{region '#Template'}
	{attribute 'Version' := '5.1.0.0'}
	{attribute 'Tags' := '"LCID": "1031", "Text": "RA, HC, Controller"'}
	{attribute 'Tags' := '"LCID": "1033", "Text": "RA, HC, Controller"'}
	{attribute 'Using' := '"Type": "Template", "URI": "BA2_Param"'}
	{attribute 'Description' := '"LCID": "1031", "Text": "Heiz-/Kühlregelung Raum"'}
	{attribute 'Description' := '"LCID": "1033", "Text": "Heating-/cooling-controller room"'}
{endregion}
FUNCTION_BLOCK FB_BA_HeatCool_PID EXTENDS FB_BA_Ext_HeatCoolBase         		
VAR_INPUT    		
	bPrc							: BOOL;				// presence-detector
	bWdwCon							: BOOL;				// window-contact - TRUE = OPEN
	eMedium							: E_BA_Medium;		// actual medium when using 2-pipe-system: heating or cooling
	bDewPnt							: BOOL;				// dew-point-detector - TRUE = ALARM
	fRmT							: REAL;				// actual room-temperature
	fRmTAdj							: REAL;				// manual adjustment of room-temperature, if desired.
	stBuildingSpRmT					: ST_BA_SpRmT;		// set points for all energy levels
	eBuildingEnergyLevel			: E_BA_EnergyLvlEx;	// current energy levels
	                                                    
END_VAR             			                        
VAR_OUTPUT          	                                
	bCtrlHtgActv					: BOOL;				// controller heating is active	
	fCtrlValHtg						: REAL;				// control-value heating
	bCtrlColActv					: BOOL;				// controller cooling is active	
	fCtrlValCol						: REAL;				// control-value cooling
	eReqdMedium						: E_BA_Medium;		// requested medium
END_VAR                                                 
VAR_INPUT CONSTANT PERSISTENT                           
	ePipeSys						: E_BA_PipeSys;		// selection 2-pipe or 4-pipe system
	{attribute 'parameterUnit':= 's'}                   
	nFnctSelChgOvrDly 				: UDINT;			// switch-over-delay from heating to cooling or vice versa	
	fRmTAdjLimit					: REAL;				// positive and negative limit of room temperature adjust value
END_VAR                  		
VAR_INPUT CONSTANT
	CtrlHtg							: FB_BA_Loop;
	CtrlCol							: FB_BA_Loop;
END_VAR
VAR
	RmTAdj							: FB_BA_RmTAdj;
	EnergLvlSlcn					: FB_BA_PrioSwi_UDI04;
	SpSlcnHtg						: FB_BA_MUX_R04;
	SpSclnCol						: FB_BA_MUX_R04;
	FnctSel							: FB_BA_FnctSel;
	RmTAdjSel						: FB_BA_LastWriterWins_R04;
	fRmTAdjLimited					: REAL;		// limited room temperature adjust value
END_VAR
VAR // added by the converter: edge detectors and wires of the graphical bodies
    _w1 : REAL;
END_VAR

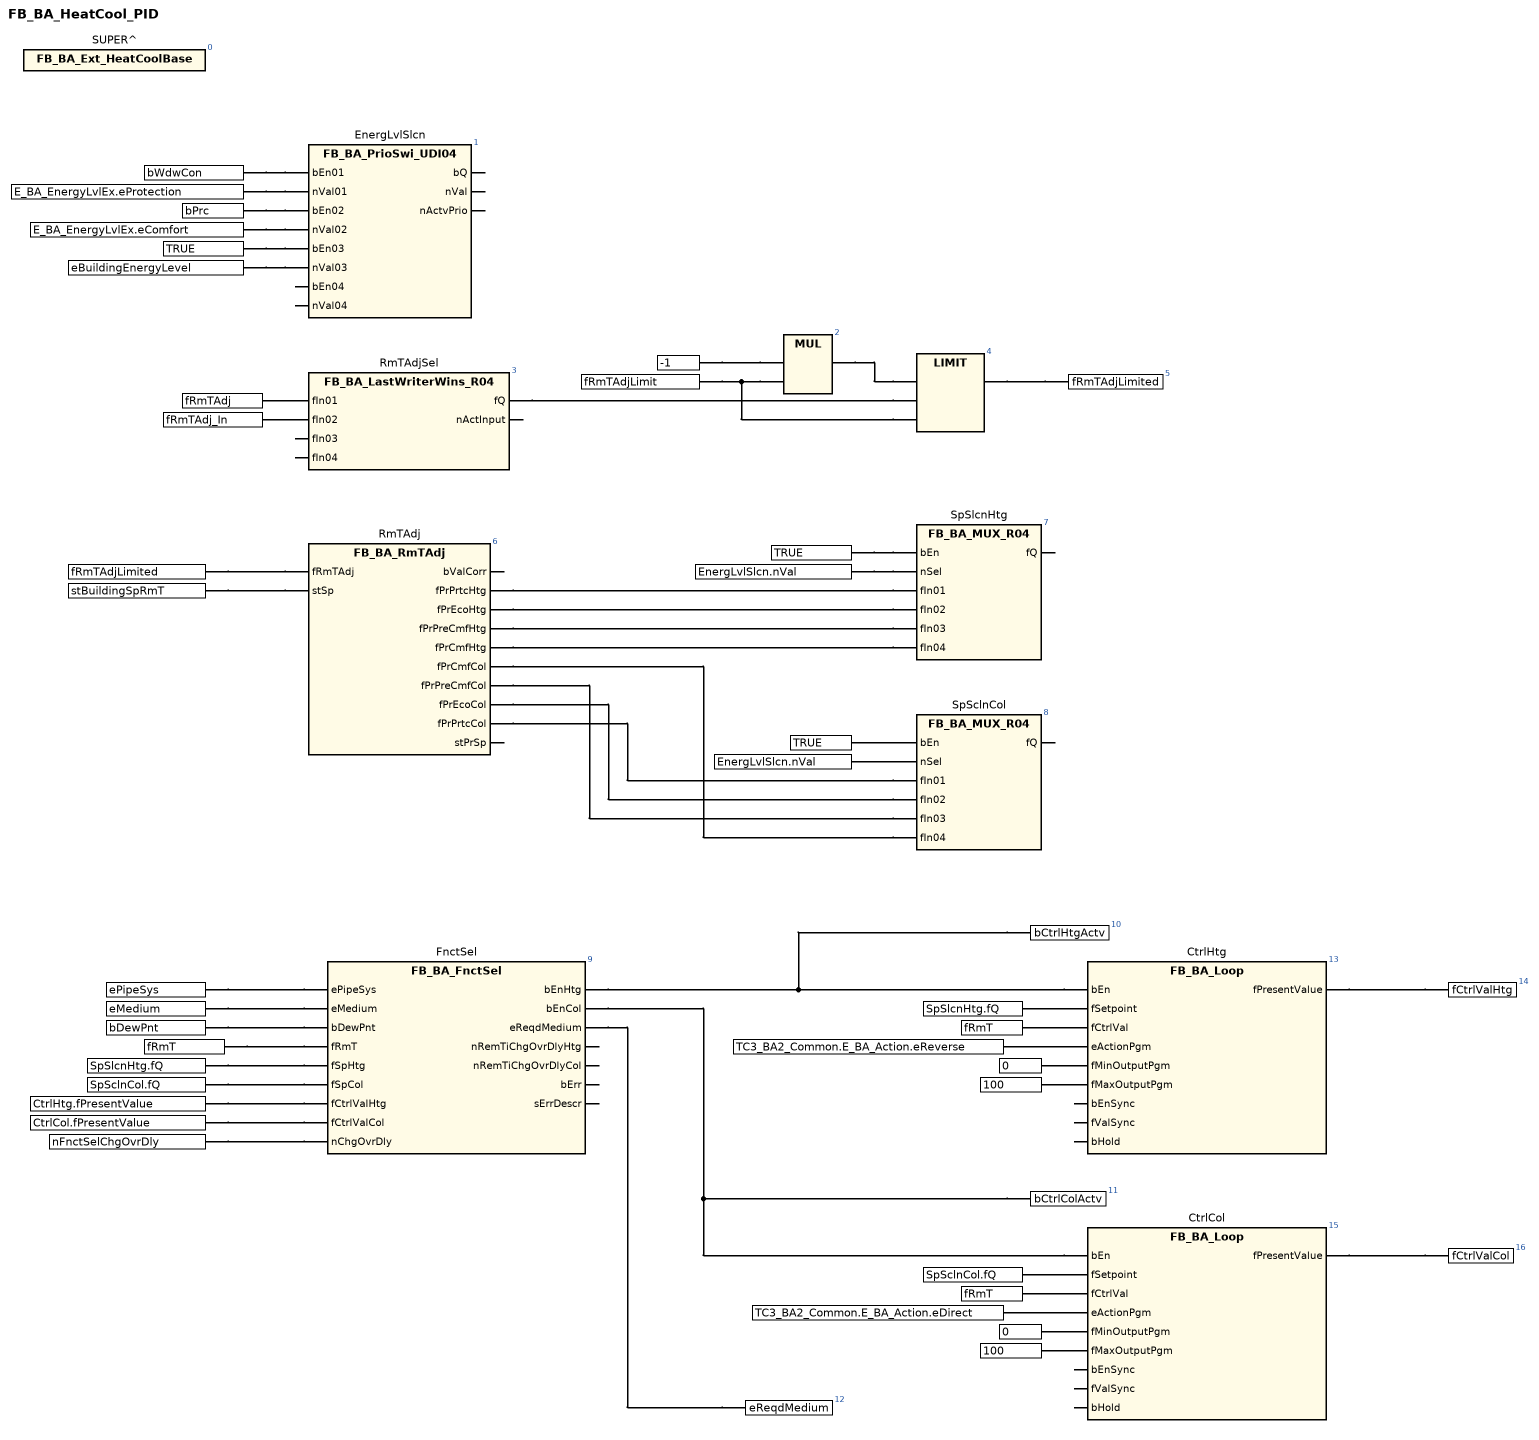
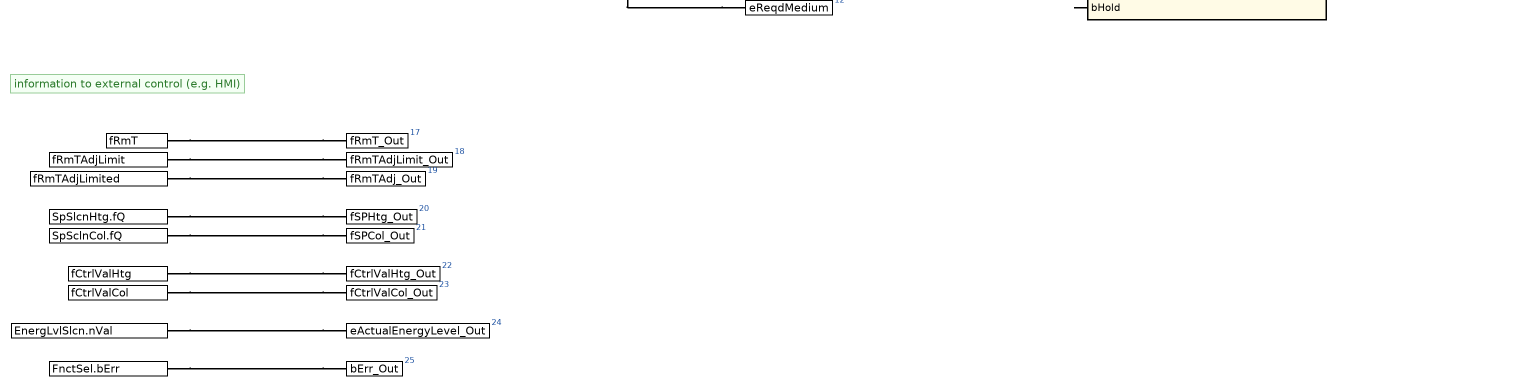
SUPER^(); // FB_BA_Ext_HeatCoolBase
EnergLvlSlcn(
    bEn01 := bWdwCon,
    nVal01 := E_BA_EnergyLvlEx.eProtection,
    bEn02 := bPrc,
    nVal02 := E_BA_EnergyLvlEx.eComfort,
    bEn03 := TRUE,
    nVal03 := eBuildingEnergyLevel); // FB_BA_PrioSwi_UDI04
_w1 := -1 * fRmTAdjLimit;
RmTAdjSel(fIn01 := fRmTAdj, fIn02 := fRmTAdj_In); // FB_BA_LastWriterWins_R04
fRmTAdjLimited := LIMIT(_w1, RmTAdjSel.fQ, fRmTAdjLimit);
RmTAdj(fRmTAdj := fRmTAdjLimited, stSp := stBuildingSpRmT); // FB_BA_RmTAdj
SpSlcnHtg(
    bEn := TRUE,
    nSel := EnergLvlSlcn.nVal,
    fIn01 := RmTAdj.fPrPrtcHtg,
    fIn02 := RmTAdj.fPrEcoHtg,
    fIn03 := RmTAdj.fPrPreCmfHtg,
    fIn04 := RmTAdj.fPrCmfHtg); // FB_BA_MUX_R04
SpSclnCol(
    bEn := TRUE,
    nSel := EnergLvlSlcn.nVal,
    fIn01 := RmTAdj.fPrPrtcCol,
    fIn02 := RmTAdj.fPrEcoCol,
    fIn03 := RmTAdj.fPrPreCmfCol,
    fIn04 := RmTAdj.fPrCmfCol); // FB_BA_MUX_R04
FnctSel(
    ePipeSys := ePipeSys,
    eMedium := eMedium,
    bDewPnt := bDewPnt,
    fRmT := fRmT,
    fSpHtg := SpSlcnHtg.fQ,
    fSpCol := SpSclnCol.fQ,
    fCtrlValHtg := CtrlHtg.fPresentValue,
    fCtrlValCol := CtrlCol.fPresentValue,
    nChgOvrDly := nFnctSelChgOvrDly); // FB_BA_FnctSel
bCtrlHtgActv := FnctSel.bEnHtg;
bCtrlColActv := FnctSel.bEnCol;
eReqdMedium := FnctSel.eReqdMedium;
CtrlHtg(
    bEn := FnctSel.bEnHtg,
    fSetpoint := SpSlcnHtg.fQ,
    fCtrlVal := fRmT,
    eActionPgm := TC3_BA2_Common.E_BA_Action.eReverse,
    fMinOutputPgm := 0,
    fMaxOutputPgm := 100); // FB_BA_Loop
fCtrlValHtg := CtrlHtg.fPresentValue;
CtrlCol(
    bEn := FnctSel.bEnCol,
    fSetpoint := SpSclnCol.fQ,
    fCtrlVal := fRmT,
    eActionPgm := TC3_BA2_Common.E_BA_Action.eDirect,
    fMinOutputPgm := 0,
    fMaxOutputPgm := 100); // FB_BA_Loop
fCtrlValCol := CtrlCol.fPresentValue;
// information to external control (e.g. HMI)
fRmT_Out := fRmT;
fRmTAdjLimit_Out := fRmTAdjLimit;
fRmTAdj_Out := fRmTAdjLimited;
fSPHtg_Out := SpSlcnHtg.fQ;
fSPCol_Out := SpSclnCol.fQ;
fCtrlValHtg_Out := fCtrlValHtg;
fCtrlValCol_Out := fCtrlValCol;
eActualEnergyLevel_Out := EnergLvlSlcn.nVal;
bErr_Out := FnctSel.bErr;

METHOD FB_init : BOOL
VAR_INPUT
	bInitRetains : BOOL; // if TRUE, the retain variables are initialized (warm start / cold start)
	bInCopyCode : BOOL;  // if TRUE, the instance afterwards gets moved into the copy code (online change)
END_VAR
ePipeSys							:= E_BA_PipeSys.e4Pipe;	// selection 2-pipe or 4-pipe system
nFnctSelChgOvrDly 					:= 120;					// switch-over-delay [s] from heating to cooling or vice versa	
fRmTAdjLimit						:= 1;					// positive and negative limit of room temperature adjust value

CtrlHtg.iParent						:= THIS^;
CtrlHtg.iLabel						:= LblCtl_RoomTemperatureControl;
CtrlHtg.eOpMode						:= E_BA_PIDMode.ePID;								 	 										 
CtrlHtg.eOutputUnit					:= E_BA_Unit.eOther_Percent;
CtrlHtg.fProportionalConstant		:= 3;
CtrlHtg.fIntegralConstant			:= 180;
CtrlHtg.fDerivativeConstant			:= 0;
CtrlHtg.fCOVIncrement				:= 0;
CtrlHtg.nDampConstant				:= 0;
CtrlHtg.fNeutralZone				:= 0;

CtrlCol.iParent						:= THIS^;
CtrlCol.iLabel						:= LblCtl_RoomTemperatureControl;
CtrlCol.eOpMode						:= E_BA_PIDMode.ePID;								 	 										 
CtrlCol.eOutputUnit					:= E_BA_Unit.eOther_Percent;
CtrlCol.fProportionalConstant		:= 3;
CtrlCol.fIntegralConstant			:= 180;
CtrlCol.fDerivativeConstant			:= 0;
CtrlCol.fCOVIncrement				:= 0;
CtrlCol.nDampConstant				:= 0;
CtrlCol.fNeutralZone				:= 0;
END_METHOD

END_FUNCTION_BLOCK

(* stored: Version 1.1.0.1, ProductVersion 3.1.4024.15
   POU FB_BA_HeatCool_PID: Id {c0e37cb5-7965-4a23-a2cd-66b383c1dd05}, SpecialFunc None
   Method FB_init: Id {7bf31459-9978-40a9-826c-a77b398eab01} *)
